{attribute 'qualified_only'}
{attribute 'strict'}
TYPE E_ModuleSequenceStatus :
(
	Idle,
	Busy,
	Waiting,
	Complete,
	Disabled,
	Error
);
END_TYPE

(* stored: Version 1.1.0.1, ProductVersion 3.1.4024.9
   DUT E_ModuleSequenceStatus: Id {07cfa4db-3828-4eb7-b3e8-5fc41ca3a46d} *)
